# EPICS autosave request: iocBoot/ioc13MeasComp2408_1/auto_settings.req
file "USB2408_settings.req",     P=$(P)
file "pid_control_settings.req"  P=$(P), PID=PID1
file "scan_settings.req",        P=$(P), S=scan1
file "scan_settings.req",        P=$(P), S=scan2
file "scan_settings.req",        P=$(P), S=scan3
file "scan_settings.req",        P=$(P), S=scan4
